Fanuc KAREL source: kc00031.KL

-- PROVISIONAL review KL for V770-1; original PC SHA256 e657a33641b4d63e74ae02629d03f6afeaa875f671c2d2599be39e071e6625b1
-- Incomplete behavior may be omitted. Consult companion uncertainty JSON. Do not deploy.
PROGRAM KC00031
%NOLOCKGROUP
BEGIN
  -- UNRESOLVED_PC offsets 5-27; opcodes 27,22,22,31,23
  -- UNRESOLVED_PC offsets 32-36; opcodes 7F
END KC00031
